FUNCTION_BLOCK Supervisor
VAR_INPUT
	EN: BOOL;
	Stop: BOOL;
END_VAR
VAR_OUTPUT
	ENO: BOOL;
END_VAR
VAR
END_VAR
VAR PERSISTENT
END_VAR

ENO := EN AND NOT Stop;

METHOD FB_init : BOOL
VAR_INPUT
	bInitRetains : BOOL; // if TRUE, the retain variables are initialized (warm start / cold start)
	bInCopyCode : BOOL;  // if TRUE, the instance afterwards gets moved into the copy code (online change)
END_VAR
END_METHOD

END_FUNCTION_BLOCK

(* stored: Version 1.1.0.1, ProductVersion 3.1.4024.3
   POU Supervisor: Id {989d1ea3-5d9d-4549-88d9-7f3bfe98bed2}, SpecialFunc None
   Method FB_init: Id {1cba1caa-cb11-4b80-ab15-4269d5e3c6b0} *)
